// TIA Portal V21 export
TYPE "Std_PausaLavoro"
   STRUCT
      Abilitazione { S7_SetPoint := 'True'} : Bool;
      DurataLavoro : "Std_stTimer";
      DurataPausa : "Std_stTimer";
   END_STRUCT;
   // DurataLavoro.IN := FALSE;
   // DurataLavoro.O := FALSE;
   // DurataLavoro.Preset := 0.0;
   // DurataLavoro.TempoTrascorso := 0.0;
   // DurataPausa.IN := FALSE;
   // DurataPausa.O := FALSE;
   // DurataPausa.Preset := 0.0;
   // DurataPausa.TempoTrascorso := 0.0;
END_TYPE
